PROGRAM MAIN
VAR
END_VAR

END_PROGRAM

(* stored: Version 1.1.0.1
   POU MAIN: Id {2305b859-3993-4f9a-8e44-5cd773bf06f0} *)
